{attribute 'pack_mode' := '1'}
TYPE
  ST_OpcUa_UintPoint EXTENDS ST_OpcUa_PointBase :
  STRUCT
    Value : UINT;
  END_STRUCT
END_TYPE

(* stored: Version 1.1.0.1, ProductVersion 3.1.4024.9
   DUT ST_OpcUa_UintPoint: Id {598db790-75f6-4efe-9343-2fc00697254f} *)
